{attribute 'no_explicit_call'}
FUNCTION_BLOCK FB_StringBuilder IMPLEMENTS I_StringBuilder
VAR_INPUT
END_VAR
VAR_OUTPUT
END_VAR
VAR
	pString:		POINTER TO STRING(1);
	aList:			POINTER TO POINTER TO STRING(1000):= ADR(pString);
	nLength:		UDINT;
END_VAR

METHOD FB_exit : BOOL
VAR_INPUT
	bInCopyCode : BOOL; // if TRUE, the exit method is called for exiting an instance that is copied afterwards (online change).
END_VAR
M_Reset();
END_METHOD

METHOD M_Append : I_StringBuilder
VAR_INPUT
	Value	: STRING(255);
END_VAR
VAR
	pValue: 	POINTER TO STRING(1):=ADR(Value);
	nValue:		UDINT:= LEN2(pValue);
	pOldList:	POINTER TO STRING(1):= pString;
END_VAR
// First Item
IF pString = 0 THEN
	nLength:= nValue;
	pString:= __NEW(STRING(1), (nLength + 1));
	CONCAT2(pString, pValue, pString, nLength + 1);
ELSE
	// new Length
	nLength:= nLength + nValue;
	// new pointer
	pString:= __NEW(STRING(1), (SIZEOF(STRING(1)) * (nLength + 1)));
	// copy to
	CONCAT2(pOldList, pValue, pString, nLength + 1);
	// delete old
	__DELETE(pOldList);

END_IF
M_Append:= THIS^;
END_METHOD

METHOD PUBLIC M_AppendBOOL  : I_StringBuilder
VAR_INPUT
	Value:			BOOL;
END_VAR
M_Append(BOOL_TO_STRING(Value));
M_AppendBOOL:= THIS^;
END_METHOD

METHOD PUBLIC M_AppendINT : I_StringBuilder
VAR_INPUT
	Value	: LINT;
END_VAR
M_Append(LINT_TO_STRING(Value));
M_AppendINT:= THIS^;
END_METHOD

METHOD PUBLIC M_AppendREAL : I_StringBuilder
VAR_INPUT
	Value:		LREAL;
	Decimals:	SINT;
END_VAR
M_Append(LREAL_TO_FMTSTR(Value, Decimals, TRUE));
M_AppendREAL:= THIS^;
END_METHOD

METHOD PUBLIC M_Contains : BOOL
VAR_INPUT
	Value	: STRING(255);
END_VAR
M_Contains:= M_Search(Value) <> 0;
END_METHOD

METHOD M_Insert : I_StringBuilder
VAR_INPUT
	Position:	UDINT;
	Value:		STRING(255);
END_VAR
VAR
	pValue: 	POINTER TO STRING(1):=ADR(Value);
	nValue:		UDINT:= LEN2(pValue);
	pOldList:	POINTER TO STRING(1):= pString;
END_VAR
IF nLength > Position AND Position <> 0 THEN
	// new Length
	nLength:= nLength + nValue;
	// new pointer
	pString:= __NEW(STRING(1), (SIZEOF(STRING(1)) * (nLength + 1)));
	// insert
	INSERT2(pOldList, pValue, pString, nLength + 1, Position -1);
	// delete old
	__DELETE(pOldList);
END_IF
M_Insert:= THIS^;
END_METHOD

METHOD M_Reset : I_StringBuilder
__DELETE(pString);
nLength:= 0;
M_Reset:= THIS^;
END_METHOD

METHOD M_Search : UDINT
VAR_INPUT
	Value	: STRING(255);
END_VAR
M_Search:= FIND2(pString, adr(Value));
END_METHOD

METHOD M_ToAny : BOOL
VAR_INPUT
	Value:			ANY;
END_VAR
Memset(Value.pValue, 0, DINT_TO_UDINT(Value.diSize));
Memcpy(Value.pValue, pString, nLength + 1);
END_METHOD

METHOD PUBLIC M_ToString : STRING(255)
VAR_INPUT
END_VAR
Memcpy(Adr(M_ToString), pString, nLength + 1);
END_METHOD

PROPERTY PUBLIC P_Length : Udint
GET
P_Length:= nLength;
END_GET
END_PROPERTY

END_FUNCTION_BLOCK

(* stored: Version 1.1.0.1
   POU FB_StringBuilder: Id {9f827a4a-fbbc-02a4-003e-5f1aba2ebf50}, SpecialFunc None
   Method FB_exit: Id {49473793-c4b9-069d-13de-b295d25dcc6b}
   Method M_Append: Id {2645d32d-7cde-0125-3686-22ccb6a7762e}
   Method M_AppendBOOL: Id {56944132-17d4-0f65-1303-77dc1a8188a8}
   Method M_AppendINT: Id {cb694219-e5bf-0cf7-0e23-ed0db5df6cae}
   Method M_AppendREAL: Id {f620367a-1ee6-014d-1c74-6ebffa68edce}
   Method M_Contains: Id {c67d02ab-f387-0562-19e3-1fdf809d8c84}
   Method M_Insert: Id {67f710af-d9b9-0cd0-2ba2-399c2edf9c98}
   Method M_Reset: Id {fc3baabb-d4a7-08e7-3d21-7dd7a233d0d0}
   Method M_Search: Id {bdf827ee-cb2f-0b2a-285b-3c9de78c6af6}
   Method M_ToAny: Id {e82dfe86-f804-0621-2a01-a384fa38ed4a}
   Method M_ToString: Id {a3197c03-d800-0530-2d92-cfaefafd28b4}
   Property P_Length: Id {c1cb7260-e235-026d-2ee4-302b9fe78fed}
   Get Get: Id {5a02b74e-a78c-0da8-22e3-f37634962917} *)
